FUNCTION_BLOCK FB_GetMasterTs
VAR_INPUT
END_VAR
VAR_OUTPUT
	MasterTsUsec: INT :=0;
END_VAR
VAR
	prevTaskTime : ULINT;//100 ns
	nowTaskTime  : ULINT;//100 ns
	nCycles : ULINT :=0;
END_VAR

prevTaskTime := nowTaskTime;
nowTaskTime  := F_GetTaskTime();
IF nCycles>0 THEN
MasterTsUsec := ULINT_TO_INT( (nowTaskTime-prevTaskTime))/10;
END_IF
nCycles := nCycles+1;

END_FUNCTION_BLOCK

(* stored: Version 1.1.0.1, ProductVersion 3.1.4024.6
   POU FB_GetMasterTs: Id {0771b7ec-c875-475d-8663-3233f5e9cd06}, SpecialFunc None *)
